TYPE ST_UdiParametr :
STRUCT
	udiValue											:	UDINT;
	udiOldValue											:	UDINT;
	udiMinLimit											:	UDINT;
	udiMaxLimit											:	UDINT;
	udiDefault											:	UDINT;
	udiColor											:	UDINT	:=	16#FFFFAF1C;	
	wsInfoCaption										:	WSTRING(100);	
	wsCaption1											:	WSTRING(50);
	wsCaption2											:	WSTRING(50);
	bUse2caption										:	BOOL;
	wsUnit												:	WSTRING;
END_STRUCT
END_TYPE

(* stored: Version 1.1.0.1, ProductVersion 3.1.4026.13, FileIdentifier 9f262a0d025a9647c03ec134379065820637de85, FileSignature 88953bd59a8200ed53ae4ac3c6c7ea146cb327f26f523dac60850cf36c423104a5534ae99178302ad4db3dacfcf274bd4bea480fdca698bdb88e232f78b059dee2643a229977c2df254d37dcf3084828e07525b96cf9a5566f1d16014cc8ef70c5c8124e87f9f6411f7e9bddbff39df39421bd4df93f540f28472e091382ba0b4f09edfb08f1a4e685c664c6723c0ae63352772d8a8d07816b459e58ccc98e2d14c227c36ac516fca781ad2896f2dcf046256ad357ae467dc4ff30a25361d349ede903db03c1ee7039ccd2b11cd08fd1b617c06b2c7219cf6aa61731cccf66cfc5e3bb902d66020265c88d2bcb7f4519f163e39011a66291ad7bcc005b6a7921
   DUT ST_UdiParametr: Id {613adb9a-a953-4e1b-ab36-3e8ff213d678} *)
